{attribute 'qualified_only'}
{attribute 'strict'}
{attribute 'to_string'}
TYPE E_CameraDevice :
(
  SheetDetect              := 0,   // SheetDetect
  PrintMark                := 1,   // PrintMark
  Scanner                  := 2,   // Scanner
  ScannerWithoutBackground := 3    // ScannerWithoutBackground
);
END_TYPE

(* stored: Version 1.1.0.1, ProductVersion 3.1.4024.3
   DUT E_CameraDevice: Id {0bb36591-9105-44b8-8600-909590b846e0} *)
